Universal Robots URScript: 00C_05_Che_BoXian.script

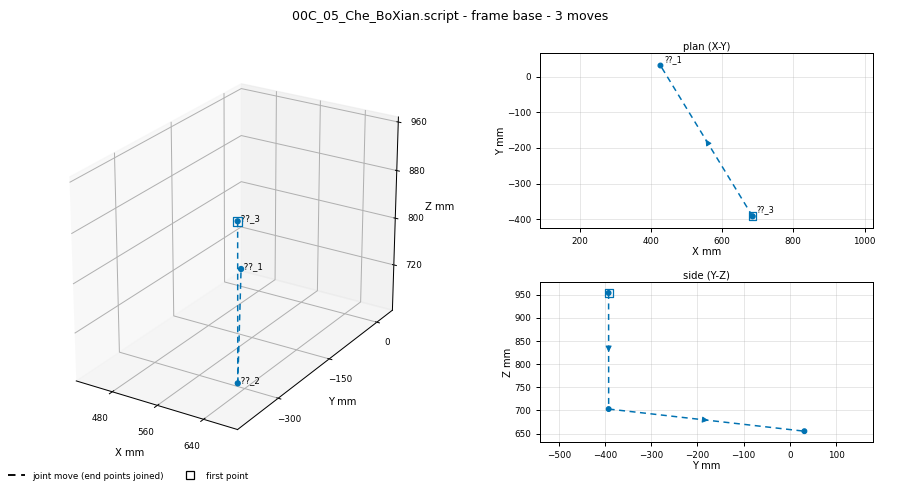
[picture p0: tool path of 00C_05_Che_BoXian.script in frame base, 3 of 3 moves have a stored position in this frame; points joined in program order, loops and branches not executed]
def P00C_05_Che_BoXian():
  set_standard_analog_input_domain(0, 1)
  set_standard_analog_input_domain(1, 1)
  set_tool_analog_input_domain(0, 1)
  set_tool_analog_input_domain(1, 1)
  set_analog_outputdomain(0, 0)
  set_analog_outputdomain(1, 0)
  set_tool_voltage(0)
  set_input_actions_to_default()
  set_tcp(p[-0.06448999999999999,0.0207,0.28314999999999996,0.0,0.0,1.5902])
  set_payload(8.0)
  set_safety_mode_transition_hardness(1)
  set_gravity([0.0, 0.0, 9.82])
  $ 1 "机器人程序"
  $ 2 "MoveJ"
  $ 3 "路点_3"
  set_tcp(p[-8.5E-4,0.01448,0.31003,0.0,0.0,-0.3645])
  movej(get_inverse_kin(p[.685511963801, -.392194506767, .954153622964, -.014200196749, .061708370629, -1.493983813725], qnear=[-0.3268993536578577, -1.7050188223468226, -1.7461841742144983, -1.3164342085467737, -1.5683091322528284, -2.3787203470813196]), a=0.6981317007977318, v=0.5235987755982988)
  $ 4 "路点_2"
  set_tcp(p[-8.5E-4,0.01448,0.31003,0.0,0.0,-0.3645])
  movej(get_inverse_kin(p[.685533586928, -.392066383948, .702936909504, -.014194078927, .061689757052, -1.493880206365], qnear=[-0.3257716337787073, -1.9238718191729944, -1.9763487021075647, -0.8674142996417444, -1.568165127431051, -2.376333777104513]), a=0.6981317007977318, v=0.5235987755982988)
  $ 5 "路点_1"
  set_tcp(p[-8.5E-4,0.01448,0.31003,0.0,0.0,-0.3645])
  movej(get_inverse_kin(p[.426856000225, .031400757768, .655026806148, -.008063241435, .061615783471, -1.298983461542], qnear=[0.501240611076355, -1.4666350523578089, -2.670887056981222, -0.6038668791400355, -1.5242565313922327, -3.007583204899923]), a=0.6981317007977318, v=0.5235987755982988)
end
